Omron Sysmac Studio project For_Kullanimi (Sysmac Studio 1.65.0.64007, StandardProject)

# Controller new_Controller_0: NX1P2-1040DT1 version 1.69
Task PrimaryTask (priority 4, period or condition 2000): Program0

VAR_GLOBAL
    Array_Index : ARRAY[1..10] OF INT;
    i : INT;
    deneme_bit : BOOL;
END_VAR

PROGRAM Program0
VAR_EXTERNAL
    i : INT;
    Array_Index : ARRAY[1..10] OF INT;
    deneme_bit : BOOL;
END_VAR

(* Section Section0: ladder, written here as Structured Text *)

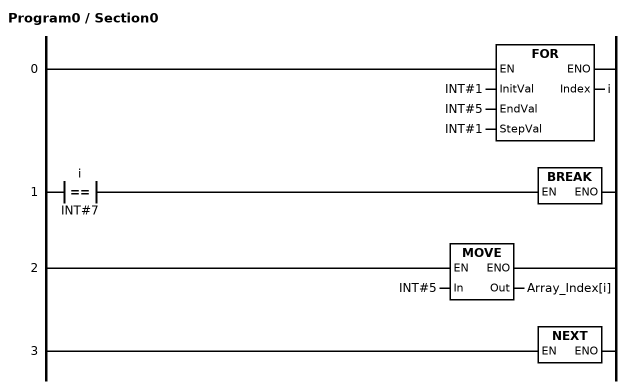
(* Rung 0 *)
i := FOR(InitVal := INT#1, EndVal := INT#5, StepVal := INT#1);
(* Rung 1 *)
IF i = INT#7 THEN BREAK(); END_IF;
(* Rung 2 *)
Array_Index[i] := INT#5;
(* Rung 3 *)
NEXT();
END_PROGRAM